Universal Robots PolyScope program: Synchronized_SpotTaping2Op.urp

Program Synchronized_SpotTaping2Op (installation=Synchronized_SpotTaping2Op directory=/home/cobot/ursim-5.11.5.1010327/programs createdIn=5.11.5.1010327 lastSavedIn=5.11.5.1010327 robotSerialNumber=20195599999)
Calibrated DH parameters: a=[0, -0.425, -0.3922, 0, 0, 0]; d=[0.1625, 0, 0, 0.1333, 0.0997, 0.0996]; alpha=[1.570796, 0, 0, 1.570796, -1.570796, 0]; deltaTheta=[0, 0, 0, 0, 0, 0]
Robot Program (runOnlyOnce=false)
  Wait DigitalInput pin=GP_bool_in[64]; digitalValue=1
  Pos1 := p[if24_x,if25_y,if26_z,GP_float_in[27],GP_float_in[28],GP_float_in[29]]
  Switch expression=GP_int_in[25]
    Case (caseValue=1)
      MoveL speed 250 mm/s, acceleration 1200 mm/s^2 (useActiveTCP=false) tcp=TCP; feature=Workspace2
        Waypoint Waypoint (Variable): variable=Pos1
    Case (caseValue=2147483647)
      MoveL speed 250 mm/s, acceleration 1200 mm/s^2 (useActiveTCP=false) tcp=TCP; feature=Workspace1
        Waypoint Waypoint (Variable): variable=Pos1
  Wait Sleep waitTime=2
  SafeHome (positionOptionType=SPEED_AND_ACCELERATION speed=1.047198 acceleration=1.396263 nextMotionTime=2)
  Set DigitalOutput pin=ob64; digitalValue=1
  Wait DigitalInput pin=ib64; digitalValue=0
  Set DigitalOutput pin=ob64; digitalValue=0
